(* PLC project Sin nombre, Desconocido Sin nombre 1 *)
(* stored: creationDateTime 2024-10-25T00:09:44, modificationDateTime 2024-10-26T19:15:56 *)

PROGRAM program0
  VAR
    timer : BOOL := 1;
    luz_1 : BOOL := 0;
    luz_2 : BOOL := 0;
    reset : BOOL := 0;
    timer_corrido_normal : BOOL := 0;
    timer_corrido_alto : BOOL := 1;
    timer_alt : BOOL := 0;
    probar_alt : BOOL := 0;
    probar_sig : BOOL := 0;
    probar_sup : BOOL := 0;
    falso : BOOL := 0;
    acumular_normal : BOOL;
    acumular_alto : BOOL;
    sal : BOOL := 0;
  END_VAR
  VAR
    sensor AT %IW0.0 : UINT := 0;
    acum AT %MW0.0 : UINT := 60000;
    acum2 AT %MW0.1 : UINT := 0;
  END_VAR
  VAR
    tope_normal : UINT := 0;
    tope_alto : UINT := 0;
    actual : INT := 3;
    TON0 : TON;
    TP1 : TP;
    TP0 : TP;
    TOF0 : TOF;
    TON1 : TON;
    TON2 : TON;
    TP2 : TP;
    TP3 : TP;
    TOF1 : TOF;
  END_VAR
  VAR  (* added by the conversion: wires and edge detectors of the diagram *)
    _ADD30_ENO : BOOL;
    _ADD30_OUT : UINT;
    _GE45_ENO : BOOL;
    _GE45_OUT : BOOL;
    _LT51_ENO : BOOL;
    _LT51_OUT : BOOL;
    _ADD67_ENO : BOOL;
    _ADD67_OUT : UINT;
    _EQ79_ENO : BOOL;
    _EQ79_OUT : BOOL;
    _LT41_ENO : BOOL;
    _LT41_OUT : BOOL;
    _GE83_ENO : BOOL;
    _GE83_OUT : BOOL;
    _ADD88_ENO : BOOL;
    _ADD88_OUT : INT;
    _EQ32_ENO : BOOL;
    _EQ32_OUT : BOOL;
    _GE55_ENO : BOOL;
    _GE55_OUT : BOOL;
    _ADD91_ENO : BOOL;
    _ADD91_OUT : INT;
    _LT97_ENO : BOOL;
    _LT97_OUT : BOOL;
  END_VAR

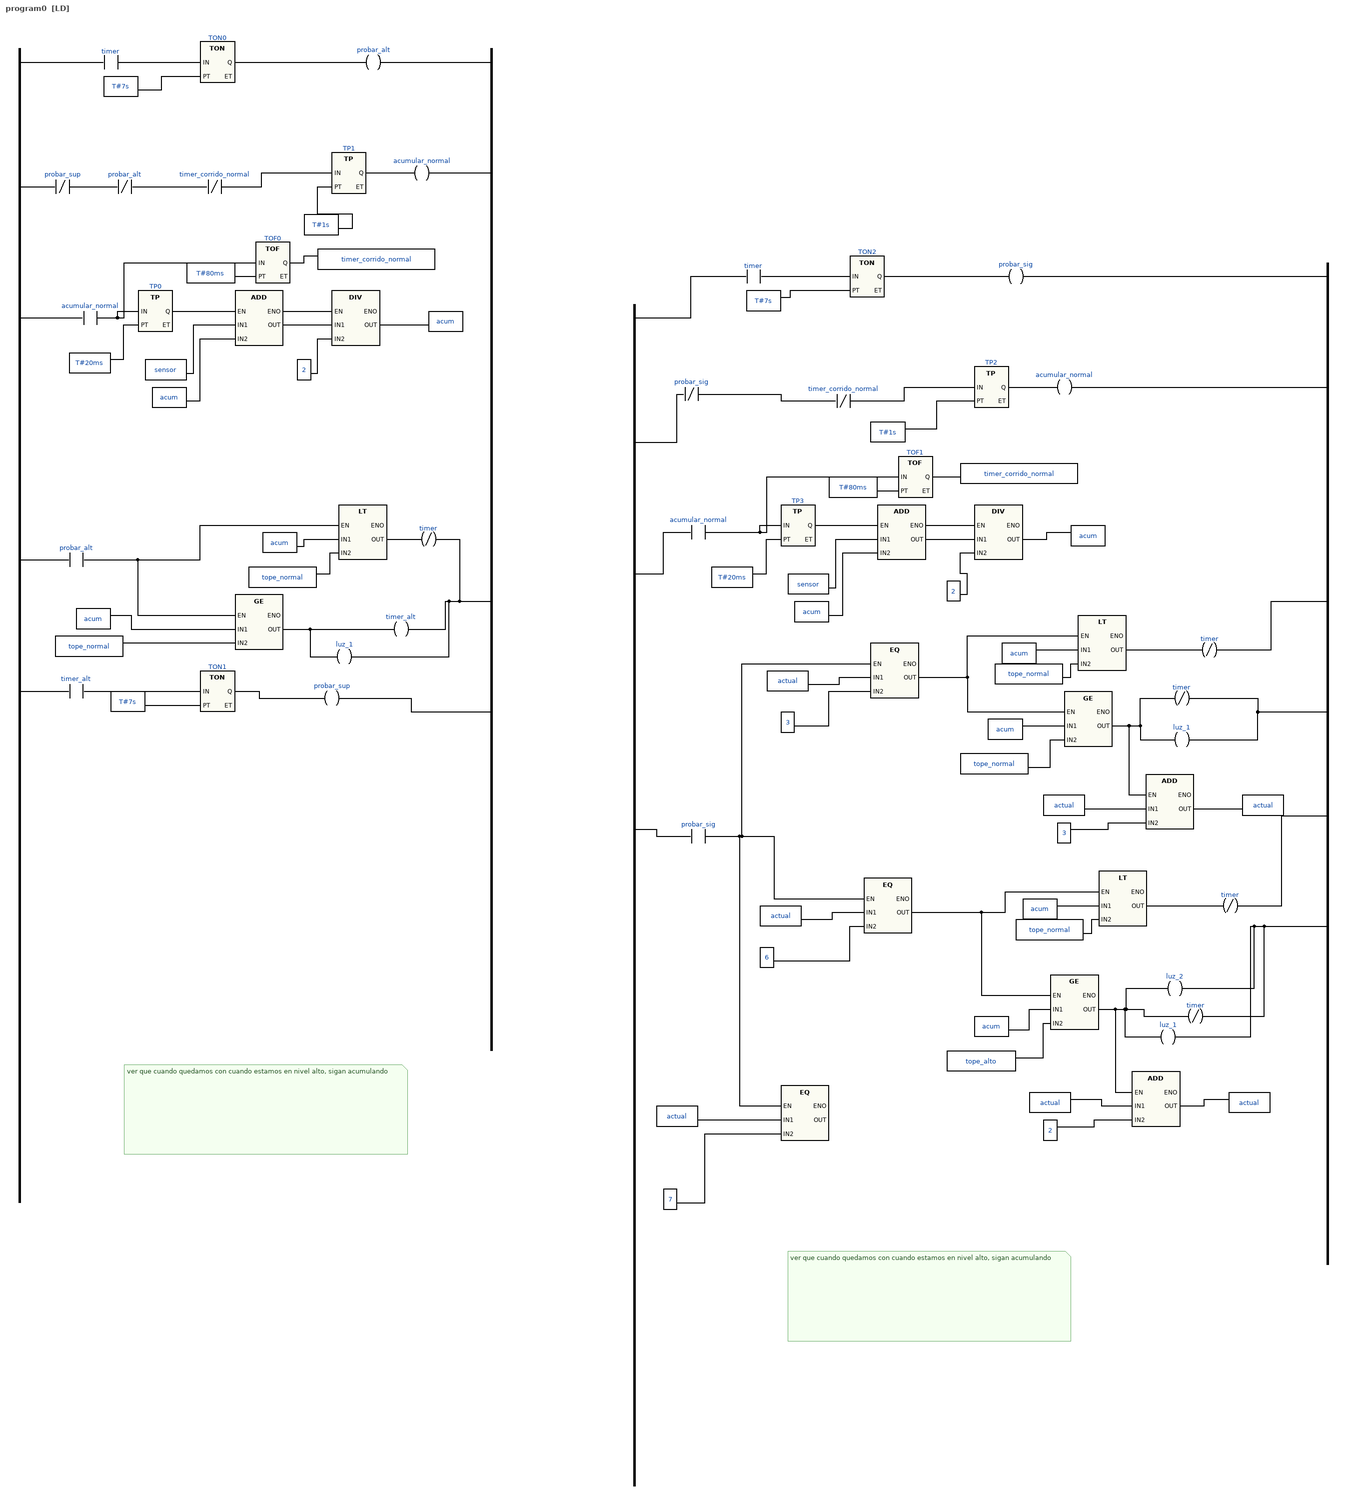
(* LD diagram, written out as Structured Text *)
TON0(IN := timer, PT := T#7s);
probar_alt := TON0.Q;
TP1(IN := NOT probar_sup AND NOT probar_alt AND NOT timer_corrido_normal, PT := T#1s);
acumular_normal := TP1.Q;
TP0(IN := acumular_normal, PT := T#20ms);
_ADD30_OUT := ADD(EN := TP0.Q, IN1 := sensor, IN2 := acum, ENO => _ADD30_ENO);
IF _ADD30_ENO THEN acum := _ADD30_OUT / 2; END_IF;
TOF0(IN := acumular_normal, PT := T#80ms);
timer_corrido_normal := TOF0.Q;
_GE45_OUT := GE(EN := probar_alt, IN1 := acum, IN2 := tope_normal, ENO => _GE45_ENO);
timer_alt := _GE45_OUT;
_LT51_OUT := LT(EN := probar_alt, IN1 := acum, IN2 := tope_normal, ENO => _LT51_ENO);
timer := NOT _LT51_OUT;
TON1(IN := timer_alt, PT := T#7s);
probar_sup := TON1.Q;
luz_1 := _GE45_OUT;
TON2(IN := timer, PT := T#7s);
probar_sig := TON2.Q;
TP2(IN := NOT probar_sig AND NOT timer_corrido_normal, PT := T#1s);
acumular_normal := TP2.Q;
TP3(IN := acumular_normal, PT := T#20ms);
_ADD67_OUT := ADD(EN := TP3.Q, IN1 := sensor, IN2 := acum, ENO => _ADD67_ENO);
IF _ADD67_ENO THEN acum := _ADD67_OUT / 2; END_IF;
TOF1(IN := acumular_normal, PT := T#80ms);
timer_corrido_normal := TOF1.Q;
_EQ79_OUT := EQ(EN := probar_sig, IN1 := actual, IN2 := 3, ENO => _EQ79_ENO);
_LT41_OUT := LT(EN := _EQ79_OUT, IN1 := acum, IN2 := tope_normal, ENO => _LT41_ENO);
timer := NOT _LT41_OUT;
_GE83_OUT := GE(EN := _EQ79_OUT, IN1 := acum, IN2 := tope_normal, ENO => _GE83_ENO);
timer := NOT _GE83_OUT;
luz_1 := _GE83_OUT;
_ADD88_OUT := ADD(EN := _GE83_OUT, IN1 := actual, IN2 := 3, ENO => _ADD88_ENO);
IF _ADD88_ENO THEN actual := _ADD88_OUT; END_IF;
_EQ32_OUT := EQ(EN := probar_sig, IN1 := actual, IN2 := 6, ENO => _EQ32_ENO);
_GE55_OUT := GE(EN := _EQ32_OUT, IN1 := acum, IN2 := tope_alto, ENO => _GE55_ENO);
luz_1 := _GE55_OUT;
(* ver que cuando quedamos con cuando estamos en nivel alto, sigan acumulando *)
_ADD91_OUT := ADD(EN := _GE55_OUT, IN1 := actual, IN2 := 2, ENO => _ADD91_ENO);
IF _ADD91_ENO THEN actual := _ADD91_OUT; END_IF;
luz_2 := _GE55_OUT;
_LT97_OUT := LT(EN := _EQ32_OUT, IN1 := acum, IN2 := tope_normal, ENO => _LT97_ENO);
timer := NOT _LT97_OUT;
timer := NOT _GE55_OUT;
IF probar_sig THEN EQ(IN1 := actual, IN2 := 7); END_IF;
(* ver que cuando quedamos con cuando estamos en nivel alto, sigan acumulando *)
END_PROGRAM

CONFIGURATION Config0
  RESOURCE Res0 ON PLC
    TASK task0(INTERVAL := T#20ms, PRIORITY := 0);
    PROGRAM instance0 WITH task0 : program0;
  END_RESOURCE
END_CONFIGURATION
